% RSLogix 500 project TIMER_TON_BAK002.RSS, saved by version 8.10.00.18 %
PROJECT "UNTITLED"    % processor: Bul.1763 MicroLogix 1100 Series B %

PROGRAM FILES
  LAD 2   4 rungs

DATA FILES
  O0 OUTPUT  4 elements
  I1 INPUT  6 elements
  S2 STATUS  66 elements
  B3 BINARY  1 elements
  T4 TIMER  2 elements
  C5 COUNTER  1 elements
  R6 CONTROL  1 elements
  N7 INTEGER  1 elements
  F8 FLOAT  1 elements

LADDER 2
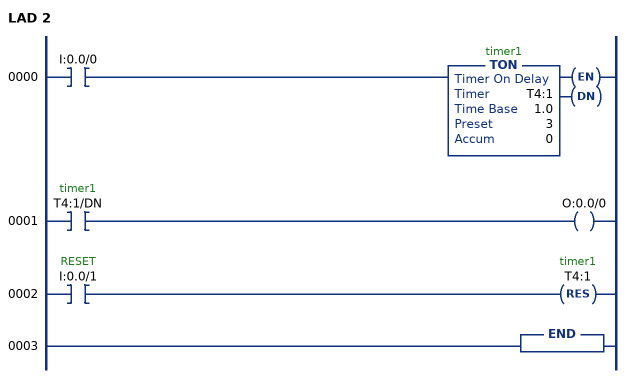
% Rung: 0 %
SOR XIC I:0.0/0 TON T4:1 1.0 3 0 EOR
%   XIC I:0.0/0  "init_timer" %
%   T4:1  "timer1" %
% Rung: 1 %
SOR XIC T4:1/DN OTE O:0.0/0 EOR
%   T4:1  "timer1" %
% Rung: 2 %
SOR XIC I:0.0/1 RES T4:1 EOR
%   I:0.0/1  "RESET" %
%   T4:1  "timer1" %
% Rung: 3 %
SOR END EOR

DATA TABLE (non-zero values as saved)
DATA T4
% .PRE .ACC %
% T4:1 % 3 0
